// Parser ErrorCode is set when a message being parsed is invalid in some way,
// e.g. malformed Varint. Zero means no error.
{attribute 'qualified_only'}
{attribute 'strict'}
{attribute 'to_string'}
TYPE E_ParserErrorCode :
(
	NoError := S_OK,            // No Error.
    InternalError := -1,        // Internal parser error.
    MalformedVarInt := -2,      // Encountered a malformed Varint.
    InvalidDataType := -3,      // Datatype not supported, e.g. F_ParseRawInt32 -> LINT
    TruncatedMessage := -4,     // 
    InvalidUtf8 := -5,          //
    NotEnoughMem := -6,         // e.g. Array [0..15] OF BYTES but F_ReadRawBytes length is 32.
    EndOfStream := -7,          //
    NotImplemented := -999      // Not implemented yet.
) DINT := NoError;
END_TYPE

(* stored: Version 1.1.0.1
   DUT E_ParserErrorCode: Id {4e8f9653-e443-4be4-a27e-634a537de09d} *)
